// TC3 §2.3/§2.7/§8.12 adapter. Task timing is measured here from TwinCAT's
// monotonic clock; target/platform diagnostic sources inject the remaining data.
FUNCTION_BLOCK FB_TcSystemHealthProbe
VAR_OUTPUT
    Health : ST_SystemHealthInput;
END_VAR
VAR
    _last : TIME;
    _windowsTime : FB_TcWindowsTime;
    _useWindowsTime : BOOL;
    _clockFile : STRING(255);
    _clockMaximumAge : TIME := T#90S;
    _clockMaximumSyncAgeSeconds : UDINT := 7200;
    _clockMaximumOffsetUs : DINT := 1000;
    _ipc : FB_TcIpcDiagnostics;
    _useIpc : BOOL;
    {attribute 'OPC.UA.DA' := '0'}
    _pBus : POINTER TO FB_EcBusHealth;
END_VAR

;

METHOD Cyclic : BOOL
VAR_INPUT
    ExpectedCycleUs       : UDINT;
    ExternalTaskOverrun   : BOOL;
    ControllerAvailable   : BOOL;
    CpuLoadPct            : LREAL;
    MemoryAvailableMb     : UDINT;
    IpcAvailable          : BOOL;
    IpcTemperatureC       : LREAL;
    FanHealthy            : BOOL;
    StorageHealthPct      : LREAL;
    FieldbusAvailable     : BOOL;
    FieldbusMasterHealthy : BOOL;
    LostFrameCount        : UDINT;
    SlaveErrorCount       : UDINT;
    DcAvailable           : BOOL;
    DcSynchronized        : BOOL;
    TimeAvailable         : BOOL;
    TimeSynchronized      : BOOL;
    TimeSource            : STRING(32);
    TimeOffsetUs          : DINT;
    LastSyncAt            : DT;
END_VAR
VAR
    currentTime, delta : TIME;
    actualUs : UDINT;
END_VAR
currentTime := TIME();
IF _last = T#0S THEN
    Health.TaskAvailable := FALSE;
    Health.TaskCycleUs := 0;
    Health.TaskJitterUs := 0;
ELSE
    delta := currentTime - _last;
    actualUs := TIME_TO_UDINT(delta) * 1000;
    Health.TaskAvailable := TRUE;
    Health.TaskCycleUs := actualUs;
    IF actualUs >= ExpectedCycleUs THEN
        Health.TaskJitterUs := actualUs - ExpectedCycleUs;
    ELSE
        Health.TaskJitterUs := ExpectedCycleUs - actualUs;
    END_IF
END_IF
_last := currentTime;
Health.TaskOverrun := ExternalTaskOverrun;
Health.ControllerAvailable := ControllerAvailable;
Health.CpuLoadPct := CpuLoadPct;
Health.MemoryAvailableMb := MemoryAvailableMb;
Health.IpcAvailable := IpcAvailable;
Health.IpcTemperatureC := IpcTemperatureC;
Health.FanHealthy := FanHealthy;
Health.StorageHealthPct := StorageHealthPct;
Health.FieldbusAvailable := FieldbusAvailable;
Health.FieldbusMasterHealthy := FieldbusMasterHealthy;
Health.LostFrameCount := LostFrameCount;
Health.SlaveErrorCount := SlaveErrorCount;
Health.DcAvailable := DcAvailable;
Health.DcSynchronized := DcSynchronized;
Health.TimeQuality.Available := TimeAvailable;
Health.TimeQuality.Synchronized := TimeAvailable AND TimeSynchronized;
Health.TimeQuality.Source := TimeSource;
Health.TimeQuality.OffsetUs := TimeOffsetUs;
Health.TimeQuality.LastSyncAt := LastSyncAt;
Health.TimeQuality.ObservedAt := F_Now();
// Explicit inputs keep the single IPC availability meaning.
Health.FanAvailable := TRUE;
Health.StorageAvailable := TRUE;
IF _useIpc THEN
    _ipc.Cyclic();
    Health.ControllerAvailable := _ipc.ControllerAvailable;
    Health.CpuLoadPct := _ipc.CpuLoadPct;
    Health.MemoryAvailableMb := _ipc.MemoryAvailableMb;
    Health.IpcAvailable := _ipc.IpcAvailable;
    Health.IpcTemperatureC := _ipc.IpcTemperatureC;
    Health.FanAvailable := _ipc.FanAvailable;
    Health.FanHealthy := _ipc.FanHealthy;
    Health.StorageAvailable := _ipc.StorageAvailable;
    Health.StorageHealthPct := _ipc.StorageHealthPct;
END_IF
IF _pBus <> 0 THEN
    Health.FieldbusAvailable := _pBus^.MasterAvailable;
    Health.FieldbusMasterHealthy := _pBus^.MasterHealthy;
    Health.LostFrameCount := _pBus^.LostFrameCount;
    Health.SlaveErrorCount := _pBus^.SlaveErrorCount;
    Health.DcAvailable := _pBus^.MasterAvailable;
    Health.DcSynchronized := _pBus^.DcSynchronized;
END_IF
IF _useWindowsTime THEN
    _windowsTime.Cyclic(FilePath := _clockFile, PollInterval := T#10S,
        MaximumSampleAge := _clockMaximumAge,
        MaximumSyncAgeSeconds := _clockMaximumSyncAgeSeconds,
        MaximumOffsetUs := _clockMaximumOffsetUs);
    Health.TimeQuality := _windowsTime.Quality;
END_IF
GVL_FraktalTime.Current := Health.TimeQuality;
Cyclic := TRUE;
END_METHOD

// Enable once at composition on a Beckhoff IPC/CX with the Device Manager: the
// controller and IPC groups then come from FB_TcIpcDiagnostics instead of the
// explicit Cyclic inputs, each available only while it is actually measured.
METHOD M_UseIpcDiagnostics : BOOL
VAR_INPUT
    Enabled : BOOL;
END_VAR
_useIpc := Enabled;
M_UseIpcDiagnostics := TRUE;
END_METHOD

// Enable once at composition: the fieldbus and DC groups then come from this
// EtherCAT adapter's always-on master sample (state, frame and CRC counters)
// instead of the explicit Cyclic inputs. 0 returns to the explicit inputs.
METHOD M_UseEtherCatMaster : BOOL
VAR_INPUT
    pBus : POINTER TO FB_EcBusHealth;
END_VAR
_pBus := pBus;
M_UseEtherCatMaster := pBus <> 0;
END_METHOD

// Enable once at composition. Cyclic owns observation and expiry thereafter.
METHOD M_UseWindowsTime : BOOL
VAR_INPUT
    Enabled : BOOL;
    FilePath : STRING(255);
    MaximumSampleAge : TIME;
    MaximumSyncAgeSeconds : UDINT;
    MaximumOffsetUs : DINT;
END_VAR
M_UseWindowsTime := (NOT Enabled)
    OR ((FilePath <> '') AND (MaximumSampleAge >= T#1S)
        AND (MaximumSyncAgeSeconds > 0) AND (MaximumOffsetUs >= 0));
_useWindowsTime := Enabled;
_clockFile := FilePath;
_clockMaximumAge := MaximumSampleAge;
_clockMaximumSyncAgeSeconds := MaximumSyncAgeSeconds;
_clockMaximumOffsetUs := MaximumOffsetUs;
END_METHOD

END_FUNCTION_BLOCK

(* stored: Version 1.1.0.1, ProductVersion 3.1.4024.12
   POU FB_TcSystemHealthProbe: Id {345ba223-e9e5-4ad3-a079-ed19f1515224}, SpecialFunc None
   Method Cyclic: Id {0f06f042-fb73-40b5-913f-84b6372142dc}
   Method M_UseIpcDiagnostics: Id {3f6c65a9-1d28-4860-9f82-e5d477a410ac}
   Method M_UseEtherCatMaster: Id {4c524c85-5b8c-4e58-90fc-b7981021ac57}
   Method M_UseWindowsTime: Id {747a1109-9972-4615-a872-79e28ab1fde6} *)
